// TIA Portal project "Progetto1" (V15.1)

(* hardware
DEVICE "S7-1200 station_1"  S7-1200 Station
   slot 0: "Telaio di montaggio_0"  S7-1200 Rack  Rack  V1.0
   slot 1: "PLC_1"  CPU 1214C DC/DC/DC  6ES7 214-1AG40-0XB0  V4.2
*)

// ===== PLC "PLC_1"  CPU 1214C DC/DC/DC =====

VAR_GLOBAL   // PLC tag table "Tabella delle variabili standard"
   "Manuale" AT %I0.3 : Bool;
   "Reset" AT %I0.4 : Bool;
   "FD1" AT %I0.0 : Bool;
   "FD2" AT %I0.1 : Bool;
   "FD3" AT %I0.2 : Bool;
   "Sirena" AT %Q0.0 : Bool;
   "Indicatore Luminoso" AT %Q0.1 : Bool;
END_VAR

ORGANIZATION_BLOCK "Main"   // OB1, LAD, ProgramCycle
TITLE = "Main Program Sweep (Cycle)"
{ S7_Optimized_Access := 'TRUE' }
VERSION : 0.1
   VAR_INPUT
      Initial_Call : Bool;   // Initial call of this OB
      Remanence : Bool;   // =True, if remanent data are available
   END_VAR
BEGIN

REGION Network 1
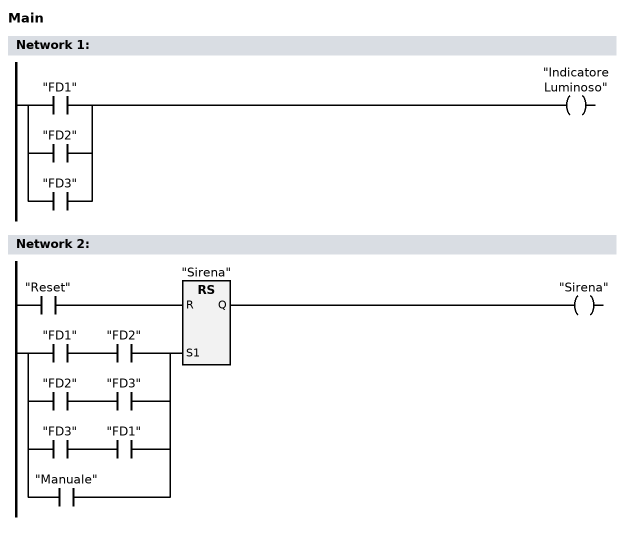
   RUNG wire#powerrail
      Contact( "FD1" )
      wire#w1
      Coil( "Indicatore Luminoso" )
   END_RUNG
   RUNG wire#powerrail
      Contact( "FD2" )
   END_RUNG wire#w1
   RUNG wire#powerrail
      Contact( "FD3" )
   END_RUNG wire#w1
   // the same network as SCL:
   "Indicatore Luminoso" := "FD1" OR "FD2" OR "FD3";
END_REGION

REGION Network 2
   RUNG wire#powerrail
      Contact( "Reset" )
      S_RS(operand := "Sirena", s1 := wire#w1)
      Coil( "Sirena" )
   END_RUNG
   RUNG wire#powerrail
      Contact( "FD1" )
      Contact( "FD2" )
   END_RUNG wire#w1
   RUNG wire#powerrail
      Contact( "FD2" )
      Contact( "FD3" )
   END_RUNG wire#w1
   RUNG wire#powerrail
      Contact( "FD3" )
      Contact( "FD1" )
   END_RUNG wire#w1
   RUNG wire#powerrail
      Contact( "Manuale" )
   END_RUNG wire#w1
   // the same network as SCL:
   IF "Reset" THEN
       "Sirena" := FALSE;   // RS flip-flop
   END_IF;
   IF ("FD1" AND "FD2") OR ("FD2" AND "FD3") OR ("FD3" AND "FD1") OR "Manuale" THEN "Sirena" := TRUE; END_IF;
   "Sirena" := "Sirena";
END_REGION
END_ORGANIZATION_BLOCK